; END LAYER 44
LIN {X -34.33, Y -49.21, Z 90.0, A 0, B 90, C 0} C_DIS
WAIT SEC 3
LIN {X -34.33, Y -49.21, Z 92.0, A 0, B 90, C 0} C_DIS
$OUT[1] = TRUE
WAIT SEC 0.8
LIN {X -34.33, Y -49.21, Z 92.0, A 0, B 90, C 0} C_DIS
LIN {X -34.33, Y -49.21, Z 92.0, A 0, B 90, C 0} C_DIS
LIN {X -31.75, Y -50.89, Z 92.0, A 0, B 90, C 0} C_DIS
LIN {X -31.1, Y -51.31, Z 92.0, A 0, B 90, C 0} C_DIS
LIN {X -28.42, Y -52.82, Z 92.0, A 0, B 90, C 0} C_DIS
LIN {X -27.75, Y -53.2, Z 92.0, A 0, B 90, C 0} C_DIS
LIN {X -24.98, Y -54.53, Z 92.0, A 0, B 90, C 0} C_DIS
LIN {X -24.29, Y -54.86, Z 92.0, A 0, B 90, C 0} C_DIS
LIN {X -21.43, Y -56.02, Z 92.0, A 0, B 90, C 0} C_DIS
LIN {X -20.72, Y -56.31, Z 92.0, A 0, B 90, C 0} C_DIS
LIN {X -17.8, Y -57.28, Z 92.0, A 0, B 90, C 0} C_DIS
LIN {X -17.07, Y -57.52, Z 92.0, A 0, B 90, C 0} C_DIS
LIN {X -14.1, Y -58.3, Z 92.0, A 0, B 90, C 0} C_DIS
LIN {X -13.35, Y -58.5, Z 92.0, A 0, B 90, C 0} C_DIS
LIN {X -10.33, Y -59.08, Z 92.0, A 0, B 90, C 0} C_DIS
LIN {X -9.58, Y -59.23, Z 92.0, A 0, B 90, C 0} C_DIS
LIN {X -6.52, Y -59.62, Z 92.0, A 0, B 90, C 0} C_DIS
LIN {X -5.76, Y -59.72, Z 92.0, A 0, B 90, C 0} C_DIS
LIN {X -2.69, Y -59.92, Z 92.0, A 0, B 90, C 0} C_DIS
LIN {X -1.92, Y -59.97, Z 92.0, A 0, B 90, C 0} C_DIS
LIN {X 1.15, Y -59.97, Z 92.0, A 0, B 90, C 0} C_DIS
LIN {X 1.92, Y -59.97, Z 92.0, A 0, B 90, C 0} C_DIS
LIN {X 4.99, Y -59.77, Z 92.0, A 0, B 90, C 0} C_DIS
LIN {X 5.76, Y -59.72, Z 92.0, A 0, B 90, C 0} C_DIS
LIN {X 8.81, Y -59.33, Z 92.0, A 0, B 90, C 0} C_DIS
LIN {X 9.58, Y -59.23, Z 92.0, A 0, B 90, C 0} C_DIS
LIN {X 12.6, Y -58.64, Z 92.0, A 0, B 90, C 0} C_DIS
LIN {X 13.35, Y -58.5, Z 92.0, A 0, B 90, C 0} C_DIS
LIN {X 16.33, Y -57.72, Z 92.0, A 0, B 90, C 0} C_DIS
LIN {X 17.07, Y -57.52, Z 92.0, A 0, B 90, C 0} C_DIS
LIN {X 19.99, Y -56.55, Z 92.0, A 0, B 90, C 0} C_DIS
LIN {X 20.72, Y -56.31, Z 92.0, A 0, B 90, C 0} C_DIS
LIN {X 23.57, Y -55.15, Z 92.0, A 0, B 90, C 0} C_DIS
LIN {X 24.29, Y -54.86, Z 92.0, A 0, B 90, C 0} C_DIS
LIN {X 27.06, Y -53.53, Z 92.0, A 0, B 90, C 0} C_DIS
LIN {X 27.75, Y -53.2, Z 92.0, A 0, B 90, C 0} C_DIS
LIN {X 30.43, Y -51.69, Z 92.0, A 0, B 90, C 0} C_DIS
LIN {X 31.1, Y -51.31, Z 92.0, A 0, B 90, C 0} C_DIS
LIN {X 33.68, Y -49.63, Z 92.0, A 0, B 90, C 0} C_DIS
LIN {X 34.33, Y -49.21, Z 92.0, A 0, B 90, C 0} C_DIS
LIN {X 36.79, Y -47.37, Z 92.0, A 0, B 90, C 0} C_DIS
LIN {X 37.41, Y -46.91, Z 92.0, A 0, B 90, C 0} C_DIS
LIN {X 39.75, Y -44.92, Z 92.0, A 0, B 90, C 0} C_DIS
LIN {X 40.34, Y -44.42, Z 92.0, A 0, B 90, C 0} C_DIS
LIN {X 42.55, Y -42.28, Z 92.0, A 0, B 90, C 0} C_DIS
LIN {X 43.1, Y -41.74, Z 92.0, A 0, B 90, C 0} C_DIS
LIN {X 45.17, Y -39.46, Z 92.0, A 0, B 90, C 0} C_DIS
LIN {X 45.69, Y -38.89, Z 92.0, A 0, B 90, C 0} C_DIS
LIN {X 47.61, Y -36.49, Z 92.0, A 0, B 90, C 0} C_DIS
LIN {X 48.08, Y -35.89, Z 92.0, A 0, B 90, C 0} C_DIS
LIN {X 49.85, Y -33.36, Z 92.0, A 0, B 90, C 0} C_DIS
LIN {X 50.29, Y -32.73, Z 92.0, A 0, B 90, C 0} C_DIS
LIN {X 51.88, Y -30.1, Z 92.0, A 0, B 90, C 0} C_DIS
LIN {X 52.28, Y -29.44, Z 92.0, A 0, B 90, C 0} C_DIS
LIN {X 53.7, Y -26.72, Z 92.0, A 0, B 90, C 0} C_DIS
LIN {X 54.06, Y -26.03, Z 92.0, A 0, B 90, C 0} C_DIS
LIN {X 55.3, Y -23.22, Z 92.0, A 0, B 90, C 0} C_DIS
LIN {X 55.62, Y -22.52, Z 92.0, A 0, B 90, C 0} C_DIS
LIN {X 56.68, Y -19.63, Z 92.0, A 0, B 90, C 0} C_DIS
LIN {X 56.94, Y -18.91, Z 92.0, A 0, B 90, C 0} C_DIS
LIN {X 57.82, Y -15.96, Z 92.0, A 0, B 90, C 0} C_DIS
LIN {X 58.04, Y -15.22, Z 92.0, A 0, B 90, C 0} C_DIS
LIN {X 58.72, Y -12.22, Z 92.0, A 0, B 90, C 0} C_DIS
LIN {X 58.89, Y -11.47, Z 92.0, A 0, B 90, C 0} C_DIS
LIN {X 59.38, Y -8.43, Z 92.0, A 0, B 90, C 0} C_DIS
LIN {X 59.51, Y -7.67, Z 92.0, A 0, B 90, C 0} C_DIS
LIN {X 59.8, Y -4.61, Z 92.0, A 0, B 90, C 0} C_DIS
LIN {X 59.88, Y -3.84, Z 92.0, A 0, B 90, C 0} C_DIS
LIN {X 59.98, Y -0.77, Z 92.0, A 0, B 90, C 0} C_DIS
LIN {X 60.0, Y -0.0, Z 92.0, A 0, B 90, C 0} C_DIS
LIN {X 59.9, Y 3.08, Z 92.0, A 0, B 90, C 0} C_DIS
LIN {X 59.88, Y 3.84, Z 92.0, A 0, B 90, C 0} C_DIS
LIN {X 59.58, Y 6.91, Z 92.0, A 0, B 90, C 0} C_DIS
LIN {X 59.51, Y 7.67, Z 92.0, A 0, B 90, C 0} C_DIS
LIN {X 59.02, Y 10.71, Z 92.0, A 0, B 90, C 0} C_DIS
LIN {X 58.89, Y 11.47, Z 92.0, A 0, B 90, C 0} C_DIS
LIN {X 58.21, Y 14.47, Z 92.0, A 0, B 90, C 0} C_DIS
LIN {X 58.04, Y 15.22, Z 92.0, A 0, B 90, C 0} C_DIS
LIN {X 57.16, Y 18.17, Z 92.0, A 0, B 90, C 0} C_DIS
LIN {X 56.94, Y 18.91, Z 92.0, A 0, B 90, C 0} C_DIS
LIN {X 55.88, Y 21.79, Z 92.0, A 0, B 90, C 0} C_DIS
LIN {X 55.62, Y 22.52, Z 92.0, A 0, B 90, C 0} C_DIS
LIN {X 54.37, Y 25.33, Z 92.0, A 0, B 90, C 0} C_DIS
LIN {X 54.06, Y 26.03, Z 92.0, A 0, B 90, C 0} C_DIS
LIN {X 52.63, Y 28.76, Z 92.0, A 0, B 90, C 0} C_DIS
LIN {X 52.28, Y 29.44, Z 92.0, A 0, B 90, C 0} C_DIS
LIN {X 50.68, Y 32.07, Z 92.0, A 0, B 90, C 0} C_DIS
LIN {X 50.29, Y 32.73, Z 92.0, A 0, B 90, C 0} C_DIS
LIN {X 48.52, Y 35.26, Z 92.0, A 0, B 90, C 0} C_DIS
LIN {X 48.08, Y 35.89, Z 92.0, A 0, B 90, C 0} C_DIS
LIN {X 46.17, Y 38.29, Z 92.0, A 0, B 90, C 0} C_DIS
LIN {X 45.69, Y 38.89, Z 92.0, A 0, B 90, C 0} C_DIS
LIN {X 43.62, Y 41.17, Z 92.0, A 0, B 90, C 0} C_DIS
LIN {X 43.1, Y 41.74, Z 92.0, A 0, B 90, C 0} C_DIS
LIN {X 40.89, Y 43.88, Z 92.0, A 0, B 90, C 0} C_DIS
LIN {X 40.34, Y 44.42, Z 92.0, A 0, B 90, C 0} C_DIS
LIN {X 38.0, Y 46.41, Z 92.0, A 0, B 90, C 0} C_DIS
LIN {X 37.41, Y 46.91, Z 92.0, A 0, B 90, C 0} C_DIS
LIN {X 34.94, Y 48.75, Z 92.0, A 0, B 90, C 0} C_DIS
LIN {X 34.33, Y 49.21, Z 92.0, A 0, B 90, C 0} C_DIS
LIN {X 31.75, Y 50.89, Z 92.0, A 0, B 90, C 0} C_DIS
LIN {X 31.1, Y 51.31, Z 92.0, A 0, B 90, C 0} C_DIS
LIN {X 28.42, Y 52.82, Z 92.0, A 0, B 90, C 0} C_DIS
LIN {X 27.75, Y 53.2, Z 92.0, A 0, B 90, C 0} C_DIS
LIN {X 24.98, Y 54.53, Z 92.0, A 0, B 90, C 0} C_DIS
LIN {X 24.29, Y 54.86, Z 92.0, A 0, B 90, C 0} C_DIS
LIN {X 21.43, Y 56.02, Z 92.0, A 0, B 90, C 0} C_DIS
LIN {X 20.72, Y 56.31, Z 92.0, A 0, B 90, C 0} C_DIS
LIN {X 17.8, Y 57.28, Z 92.0, A 0, B 90, C 0} C_DIS
LIN {X 17.07, Y 57.52, Z 92.0, A 0, B 90, C 0} C_DIS
LIN {X 14.1, Y 58.3, Z 92.0, A 0, B 90, C 0} C_DIS
LIN {X 13.35, Y 58.5, Z 92.0, A 0, B 90, C 0} C_DIS
LIN {X 10.33, Y 59.08, Z 92.0, A 0, B 90, C 0} C_DIS
LIN {X 9.58, Y 59.23, Z 92.0, A 0, B 90, C 0} C_DIS
LIN {X 6.52, Y 59.62, Z 92.0, A 0, B 90, C 0} C_DIS
LIN {X 5.76, Y 59.72, Z 92.0, A 0, B 90, C 0} C_DIS
LIN {X 2.69, Y 59.92, Z 92.0, A 0, B 90, C 0} C_DIS
LIN {X 1.92, Y 59.97, Z 92.0, A 0, B 90, C 0} C_DIS
LIN {X -1.15, Y 59.97, Z 92.0, A 0, B 90, C 0} C_DIS
LIN {X -1.92, Y 59.97, Z 92.0, A 0, B 90, C 0} C_DIS
LIN {X -4.99, Y 59.77, Z 92.0, A 0, B 90, C 0} C_DIS
LIN {X -5.76, Y 59.72, Z 92.0, A 0, B 90, C 0} C_DIS
LIN {X -8.81, Y 59.33, Z 92.0, A 0, B 90, C 0} C_DIS
LIN {X -9.58, Y 59.23, Z 92.0, A 0, B 90, C 0} C_DIS
LIN {X -12.6, Y 58.64, Z 92.0, A 0, B 90, C 0} C_DIS
LIN {X -13.35, Y 58.5, Z 92.0, A 0, B 90, C 0} C_DIS
LIN {X -16.33, Y 57.72, Z 92.0, A 0, B 90, C 0} C_DIS
LIN {X -17.07, Y 57.52, Z 92.0, A 0, B 90, C 0} C_DIS
LIN {X -19.99, Y 56.55, Z 92.0, A 0, B 90, C 0} C_DIS
LIN {X -20.72, Y 56.31, Z 92.0, A 0, B 90, C 0} C_DIS
LIN {X -23.57, Y 55.15, Z 92.0, A 0, B 90, C 0} C_DIS
LIN {X -24.29, Y 54.86, Z 92.0, A 0, B 90, C 0} C_DIS
LIN {X -27.06, Y 53.53, Z 92.0, A 0, B 90, C 0} C_DIS
LIN {X -27.75, Y 53.2, Z 92.0, A 0, B 90, C 0} C_DIS
LIN {X -30.43, Y 51.69, Z 92.0, A 0, B 90, C 0} C_DIS
LIN {X -31.1, Y 51.31, Z 92.0, A 0, B 90, C 0} C_DIS
LIN {X -33.68, Y 49.63, Z 92.0, A 0, B 90, C 0} C_DIS
LIN {X -34.33, Y 49.21, Z 92.0, A 0, B 90, C 0} C_DIS
LIN {X -36.79, Y 47.37, Z 92.0, A 0, B 90, C 0} C_DIS
LIN {X -37.41, Y 46.91, Z 92.0, A 0, B 90, C 0} C_DIS
LIN {X -39.75, Y 44.92, Z 92.0, A 0, B 90, C 0} C_DIS
LIN {X -40.34, Y 44.42, Z 92.0, A 0, B 90, C 0} C_DIS
LIN {X -42.55, Y 42.28, Z 92.0, A 0, B 90, C 0} C_DIS
LIN {X -43.1, Y 41.74, Z 92.0, A 0, B 90, C 0} C_DIS
LIN {X -45.17, Y 39.46, Z 92.0, A 0, B 90, C 0} C_DIS
LIN {X -45.69, Y 38.89, Z 92.0, A 0, B 90, C 0} C_DIS
LIN {X -47.61, Y 36.49, Z 92.0, A 0, B 90, C 0} C_DIS
LIN {X -48.08, Y 35.89, Z 92.0, A 0, B 90, C 0} C_DIS
LIN {X -49.85, Y 33.36, Z 92.0, A 0, B 90, C 0} C_DIS
LIN {X -50.29, Y 32.73, Z 92.0, A 0, B 90, C 0} C_DIS
LIN {X -51.88, Y 30.1, Z 92.0, A 0, B 90, C 0} C_DIS
LIN {X -52.28, Y 29.44, Z 92.0, A 0, B 90, C 0} C_DIS
LIN {X -53.7, Y 26.72, Z 92.0, A 0, B 90, C 0} C_DIS
LIN {X -54.06, Y 26.03, Z 92.0, A 0, B 90, C 0} C_DIS
LIN {X -55.3, Y 23.22, Z 92.0, A 0, B 90, C 0} C_DIS
LIN {X -55.62, Y 22.52, Z 92.0, A 0, B 90, C 0} C_DIS
LIN {X -56.68, Y 19.63, Z 92.0, A 0, B 90, C 0} C_DIS
LIN {X -56.94, Y 18.91, Z 92.0, A 0, B 90, C 0} C_DIS
LIN {X -57.82, Y 15.96, Z 92.0, A 0, B 90, C 0} C_DIS
LIN {X -58.04, Y 15.22, Z 92.0, A 0, B 90, C 0} C_DIS
LIN {X -58.72, Y 12.22, Z 92.0, A 0, B 90, C 0} C_DIS
LIN {X -58.89, Y 11.47, Z 92.0, A 0, B 90, C 0} C_DIS
LIN {X -59.38, Y 8.43, Z 92.0, A 0, B 90, C 0} C_DIS
LIN {X -59.51, Y 7.67, Z 92.0, A 0, B 90, C 0} C_DIS
LIN {X -59.8, Y 4.61, Z 92.0, A 0, B 90, C 0} C_DIS
LIN {X -59.88, Y 3.84, Z 92.0, A 0, B 90, C 0} C_DIS
LIN {X -59.98, Y 0.77, Z 92.0, A 0, B 90, C 0} C_DIS
LIN {X -60.0, Y -0.0, Z 92.0, A 0, B 90, C 0} C_DIS
LIN {X -59.9, Y -3.08, Z 92.0, A 0, B 90, C 0} C_DIS
LIN {X -59.88, Y -3.84, Z 92.0, A 0, B 90, C 0} C_DIS
LIN {X -59.58, Y -6.91, Z 92.0, A 0, B 90, C 0} C_DIS
LIN {X -59.51, Y -7.67, Z 92.0, A 0, B 90, C 0} C_DIS
LIN {X -59.02, Y -10.71, Z 92.0, A 0, B 90, C 0} C_DIS
LIN {X -58.89, Y -11.47, Z 92.0, A 0, B 90, C 0} C_DIS
LIN {X -58.21, Y -14.47, Z 92.0, A 0, B 90, C 0} C_DIS
LIN {X -58.04, Y -15.22, Z 92.0, A 0, B 90, C 0} C_DIS
LIN {X -57.16, Y -18.17, Z 92.0, A 0, B 90, C 0} C_DIS
LIN {X -56.94, Y -18.91, Z 92.0, A 0, B 90, C 0} C_DIS
LIN {X -55.88, Y -21.79, Z 92.0, A 0, B 90, C 0} C_DIS
LIN {X -55.62, Y -22.52, Z 92.0, A 0, B 90, C 0} C_DIS
LIN {X -54.37, Y -25.33, Z 92.0, A 0, B 90, C 0} C_DIS
LIN {X -54.06, Y -26.03, Z 92.0, A 0, B 90, C 0} C_DIS
LIN {X -52.63, Y -28.76, Z 92.0, A 0, B 90, C 0} C_DIS
LIN {X -52.28, Y -29.44, Z 92.0, A 0, B 90, C 0} C_DIS
LIN {X -50.68, Y -32.07, Z 92.0, A 0, B 90, C 0} C_DIS
LIN {X -50.29, Y -32.73, Z 92.0, A 0, B 90, C 0} C_DIS
LIN {X -48.52, Y -35.26, Z 92.0, A 0, B 90, C 0} C_DIS
LIN {X -48.08, Y -35.89, Z 92.0, A 0, B 90, C 0} C_DIS
LIN {X -46.17, Y -38.29, Z 92.0, A 0, B 90, C 0} C_DIS
LIN {X -45.69, Y -38.89, Z 92.0, A 0, B 90, C 0} C_DIS
LIN {X -43.62, Y -41.17, Z 92.0, A 0, B 90, C 0} C_DIS
LIN {X -43.1, Y -41.74, Z 92.0, A 0, B 90, C 0} C_DIS
LIN {X -40.89, Y -43.88, Z 92.0, A 0, B 90, C 0} C_DIS
LIN {X -40.34, Y -44.42, Z 92.0, A 0, B 90, C 0} C_DIS
LIN {X -38.0, Y -46.41, Z 92.0, A 0, B 90, C 0} C_DIS
LIN {X -37.41, Y -46.91, Z 92.0, A 0, B 90, C 0} C_DIS
LIN {X -34.94, Y -48.75, Z 92.0, A 0, B 90, C 0} C_DIS
$OUT[1] = FALSE

; END LAYER 45
LIN {X -34.33, Y -49.21, Z 92.0, A 0, B 90, C 0} C_DIS
WAIT SEC 3
LIN {X -34.33, Y -49.21, Z 94.0, A 0, B 90, C 0} C_DIS
$OUT[1] = TRUE
WAIT SEC 0.8
LIN {X -34.33, Y -49.21, Z 94.0, A 0, B 90, C 0} C_DIS
LIN {X -34.33, Y -49.21, Z 94.0, A 0, B 90, C 0} C_DIS
LIN {X -31.62, Y -50.97, Z 94.0, A 0, B 90, C 0} C_DIS
LIN {X -31.1, Y -51.31, Z 94.0, A 0, B 90, C 0} C_DIS
LIN {X -28.29, Y -52.89, Z 94.0, A 0, B 90, C 0} C_DIS
LIN {X -27.75, Y -53.2, Z 94.0, A 0, B 90, C 0} C_DIS
LIN {X -24.84, Y -54.6, Z 94.0, A 0, B 90, C 0} C_DIS
LIN {X -24.29, Y -54.86, Z 94.0, A 0, B 90, C 0} C_DIS
LIN {X -21.29, Y -56.08, Z 94.0, A 0, B 90, C 0} C_DIS
LIN {X -20.72, Y -56.31, Z 94.0, A 0, B 90, C 0} C_DIS
LIN {X -17.66, Y -57.33, Z 94.0, A 0, B 90, C 0} C_DIS
LIN {X -17.07, Y -57.52, Z 94.0, A 0, B 90, C 0} C_DIS
LIN {X -13.95, Y -58.34, Z 94.0, A 0, B 90, C 0} C_DIS
LIN {X -13.35, Y -58.5, Z 94.0, A 0, B 90, C 0} C_DIS
LIN {X -10.18, Y -59.11, Z 94.0, A 0, B 90, C 0} C_DIS
LIN {X -9.58, Y -59.23, Z 94.0, A 0, B 90, C 0} C_DIS
LIN {X -6.37, Y -59.64, Z 94.0, A 0, B 90, C 0} C_DIS
LIN {X -5.76, Y -59.72, Z 94.0, A 0, B 90, C 0} C_DIS
LIN {X -2.54, Y -59.93, Z 94.0, A 0, B 90, C 0} C_DIS
LIN {X -1.92, Y -59.97, Z 94.0, A 0, B 90, C 0} C_DIS
LIN {X 1.31, Y -59.97, Z 94.0, A 0, B 90, C 0} C_DIS
LIN {X 1.92, Y -59.97, Z 94.0, A 0, B 90, C 0} C_DIS
LIN {X 5.15, Y -59.76, Z 94.0, A 0, B 90, C 0} C_DIS
LIN {X 5.76, Y -59.72, Z 94.0, A 0, B 90, C 0} C_DIS
LIN {X 8.97, Y -59.31, Z 94.0, A 0, B 90, C 0} C_DIS
LIN {X 9.58, Y -59.23, Z 94.0, A 0, B 90, C 0} C_DIS
LIN {X 12.75, Y -58.61, Z 94.0, A 0, B 90, C 0} C_DIS
LIN {X 13.35, Y -58.5, Z 94.0, A 0, B 90, C 0} C_DIS
LIN {X 16.48, Y -57.68, Z 94.0, A 0, B 90, C 0} C_DIS
LIN {X 17.07, Y -57.52, Z 94.0, A 0, B 90, C 0} C_DIS
LIN {X 20.14, Y -56.5, Z 94.0, A 0, B 90, C 0} C_DIS
LIN {X 20.72, Y -56.31, Z 94.0, A 0, B 90, C 0} C_DIS
LIN {X 23.72, Y -55.1, Z 94.0, A 0, B 90, C 0} C_DIS
LIN {X 24.29, Y -54.86, Z 94.0, A 0, B 90, C 0} C_DIS
LIN {X 27.2, Y -53.46, Z 94.0, A 0, B 90, C 0} C_DIS
LIN {X 27.75, Y -53.2, Z 94.0, A 0, B 90, C 0} C_DIS
LIN {X 30.57, Y -51.61, Z 94.0, A 0, B 90, C 0} C_DIS
LIN {X 31.1, Y -51.31, Z 94.0, A 0, B 90, C 0} C_DIS
LIN {X 33.81, Y -49.55, Z 94.0, A 0, B 90, C 0} C_DIS
LIN {X 34.33, Y -49.21, Z 94.0, A 0, B 90, C 0} C_DIS
LIN {X 36.92, Y -47.28, Z 94.0, A 0, B 90, C 0} C_DIS
LIN {X 37.41, Y -46.91, Z 94.0, A 0, B 90, C 0} C_DIS
LIN {X 39.87, Y -44.82, Z 94.0, A 0, B 90, C 0} C_DIS
LIN {X 40.34, Y -44.42, Z 94.0, A 0, B 90, C 0} C_DIS
LIN {X 42.66, Y -42.17, Z 94.0, A 0, B 90, C 0} C_DIS
LIN {X 43.1, Y -41.74, Z 94.0, A 0, B 90, C 0} C_DIS
LIN {X 45.27, Y -39.35, Z 94.0, A 0, B 90, C 0} C_DIS
LIN {X 45.69, Y -38.89, Z 94.0, A 0, B 90, C 0} C_DIS
LIN {X 47.7, Y -36.37, Z 94.0, A 0, B 90, C 0} C_DIS
LIN {X 48.08, Y -35.89, Z 94.0, A 0, B 90, C 0} C_DIS
LIN {X 49.93, Y -33.24, Z 94.0, A 0, B 90, C 0} C_DIS
LIN {X 50.29, Y -32.73, Z 94.0, A 0, B 90, C 0} C_DIS
LIN {X 51.96, Y -29.97, Z 94.0, A 0, B 90, C 0} C_DIS
LIN {X 52.28, Y -29.44, Z 94.0, A 0, B 90, C 0} C_DIS
LIN {X 53.77, Y -26.58, Z 94.0, A 0, B 90, C 0} C_DIS
LIN {X 54.06, Y -26.03, Z 94.0, A 0, B 90, C 0} C_DIS
LIN {X 55.37, Y -23.08, Z 94.0, A 0, B 90, C 0} C_DIS
LIN {X 55.62, Y -22.52, Z 94.0, A 0, B 90, C 0} C_DIS
LIN {X 56.73, Y -19.48, Z 94.0, A 0, B 90, C 0} C_DIS
LIN {X 56.94, Y -18.91, Z 94.0, A 0, B 90, C 0} C_DIS
LIN {X 57.86, Y -15.81, Z 94.0, A 0, B 90, C 0} C_DIS
LIN {X 58.04, Y -15.22, Z 94.0, A 0, B 90, C 0} C_DIS
LIN {X 58.76, Y -12.07, Z 94.0, A 0, B 90, C 0} C_DIS
LIN {X 58.89, Y -11.47, Z 94.0, A 0, B 90, C 0} C_DIS
LIN {X 59.41, Y -8.28, Z 94.0, A 0, B 90, C 0} C_DIS
LIN {X 59.51, Y -7.67, Z 94.0, A 0, B 90, C 0} C_DIS
LIN {X 59.82, Y -4.46, Z 94.0, A 0, B 90, C 0} C_DIS
LIN {X 59.88, Y -3.84, Z 94.0, A 0, B 90, C 0} C_DIS
LIN {X 59.98, Y -0.62, Z 94.0, A 0, B 90, C 0} C_DIS
LIN {X 60.0, Y -0.0, Z 94.0, A 0, B 90, C 0} C_DIS
LIN {X 59.9, Y 3.23, Z 94.0, A 0, B 90, C 0} C_DIS
LIN {X 59.88, Y 3.84, Z 94.0, A 0, B 90, C 0} C_DIS
LIN {X 59.57, Y 7.06, Z 94.0, A 0, B 90, C 0} C_DIS
LIN {X 59.51, Y 7.67, Z 94.0, A 0, B 90, C 0} C_DIS
LIN {X 58.99, Y 10.86, Z 94.0, A 0, B 90, C 0} C_DIS
LIN {X 58.89, Y 11.47, Z 94.0, A 0, B 90, C 0} C_DIS
LIN {X 58.17, Y 14.62, Z 94.0, A 0, B 90, C 0} C_DIS
LIN {X 58.04, Y 15.22, Z 94.0, A 0, B 90, C 0} C_DIS
LIN {X 57.12, Y 18.32, Z 94.0, A 0, B 90, C 0} C_DIS
LIN {X 56.94, Y 18.91, Z 94.0, A 0, B 90, C 0} C_DIS
LIN {X 55.83, Y 21.94, Z 94.0, A 0, B 90, C 0} C_DIS
LIN {X 55.62, Y 22.52, Z 94.0, A 0, B 90, C 0} C_DIS
LIN {X 54.31, Y 25.47, Z 94.0, A 0, B 90, C 0} C_DIS
LIN {X 54.06, Y 26.03, Z 94.0, A 0, B 90, C 0} C_DIS
LIN {X 52.56, Y 28.9, Z 94.0, A 0, B 90, C 0} C_DIS
LIN {X 52.28, Y 29.44, Z 94.0, A 0, B 90, C 0} C_DIS
LIN {X 50.6, Y 32.21, Z 94.0, A 0, B 90, C 0} C_DIS
LIN {X 50.29, Y 32.73, Z 94.0, A 0, B 90, C 0} C_DIS
LIN {X 48.44, Y 35.38, Z 94.0, A 0, B 90, C 0} C_DIS
LIN {X 48.08, Y 35.89, Z 94.0, A 0, B 90, C 0} C_DIS
LIN {X 46.07, Y 38.41, Z 94.0, A 0, B 90, C 0} C_DIS
LIN {X 45.69, Y 38.89, Z 94.0, A 0, B 90, C 0} C_DIS
LIN {X 43.51, Y 41.29, Z 94.0, A 0, B 90, C 0} C_DIS
LIN {X 43.1, Y 41.74, Z 94.0, A 0, B 90, C 0} C_DIS
LIN {X 40.78, Y 43.99, Z 94.0, A 0, B 90, C 0} C_DIS
LIN {X 40.34, Y 44.42, Z 94.0, A 0, B 90, C 0} C_DIS
LIN {X 37.88, Y 46.51, Z 94.0, A 0, B 90, C 0} C_DIS
LIN {X 37.41, Y 46.91, Z 94.0, A 0, B 90, C 0} C_DIS
LIN {X 34.82, Y 48.84, Z 94.0, A 0, B 90, C 0} C_DIS
LIN {X 34.33, Y 49.21, Z 94.0, A 0, B 90, C 0} C_DIS
LIN {X 31.62, Y 50.97, Z 94.0, A 0, B 90, C 0} C_DIS
LIN {X 31.1, Y 51.31, Z 94.0, A 0, B 90, C 0} C_DIS
LIN {X 28.29, Y 52.89, Z 94.0, A 0, B 90, C 0} C_DIS
LIN {X 27.75, Y 53.2, Z 94.0, A 0, B 90, C 0} C_DIS
LIN {X 24.84, Y 54.6, Z 94.0, A 0, B 90, C 0} C_DIS
LIN {X 24.29, Y 54.86, Z 94.0, A 0, B 90, C 0} C_DIS
LIN {X 21.29, Y 56.08, Z 94.0, A 0, B 90, C 0} C_DIS
LIN {X 20.72, Y 56.31, Z 94.0, A 0, B 90, C 0} C_DIS
LIN {X 17.66, Y 57.33, Z 94.0, A 0, B 90, C 0} C_DIS
LIN {X 17.07, Y 57.52, Z 94.0, A 0, B 90, C 0} C_DIS
LIN {X 13.95, Y 58.34, Z 94.0, A 0, B 90, C 0} C_DIS
LIN {X 13.35, Y 58.5, Z 94.0, A 0, B 90, C 0} C_DIS
LIN {X 10.18, Y 59.11, Z 94.0, A 0, B 90, C 0} C_DIS
LIN {X 9.58, Y 59.23, Z 94.0, A 0, B 90, C 0} C_DIS
LIN {X 6.37, Y 59.64, Z 94.0, A 0, B 90, C 0} C_DIS
LIN {X 5.76, Y 59.72, Z 94.0, A 0, B 90, C 0} C_DIS
LIN {X 2.54, Y 59.93, Z 94.0, A 0, B 90, C 0} C_DIS
LIN {X 1.92, Y 59.97, Z 94.0, A 0, B 90, C 0} C_DIS
LIN {X -1.31, Y 59.97, Z 94.0, A 0, B 90, C 0} C_DIS
LIN {X -1.92, Y 59.97, Z 94.0, A 0, B 90, C 0} C_DIS
LIN {X -5.15, Y 59.76, Z 94.0, A 0, B 90, C 0} C_DIS
LIN {X -5.76, Y 59.72, Z 94.0, A 0, B 90, C 0} C_DIS
LIN {X -8.97, Y 59.31, Z 94.0, A 0, B 90, C 0} C_DIS
LIN {X -9.58, Y 59.23, Z 94.0, A 0, B 90, C 0} C_DIS
LIN {X -12.75, Y 58.61, Z 94.0, A 0, B 90, C 0} C_DIS
LIN {X -13.35, Y 58.5, Z 94.0, A 0, B 90, C 0} C_DIS
LIN {X -16.48, Y 57.68, Z 94.0, A 0, B 90, C 0} C_DIS
LIN {X -17.07, Y 57.52, Z 94.0, A 0, B 90, C 0} C_DIS
LIN {X -20.14, Y 56.5, Z 94.0, A 0, B 90, C 0} C_DIS
LIN {X -20.72, Y 56.31, Z 94.0, A 0, B 90, C 0} C_DIS
LIN {X -23.72, Y 55.1, Z 94.0, A 0, B 90, C 0} C_DIS
LIN {X -24.29, Y 54.86, Z 94.0, A 0, B 90, C 0} C_DIS
LIN {X -27.2, Y 53.46, Z 94.0, A 0, B 90, C 0} C_DIS
LIN {X -27.75, Y 53.2, Z 94.0, A 0, B 90, C 0} C_DIS
LIN {X -30.57, Y 51.61, Z 94.0, A 0, B 90, C 0} C_DIS
LIN {X -31.1, Y 51.31, Z 94.0, A 0, B 90, C 0} C_DIS
LIN {X -33.81, Y 49.55, Z 94.0, A 0, B 90, C 0} C_DIS
LIN {X -34.33, Y 49.21, Z 94.0, A 0, B 90, C 0} C_DIS
LIN {X -36.92, Y 47.28, Z 94.0, A 0, B 90, C 0} C_DIS
LIN {X -37.41, Y 46.91, Z 94.0, A 0, B 90, C 0} C_DIS
LIN {X -39.87, Y 44.82, Z 94.0, A 0, B 90, C 0} C_DIS
LIN {X -40.34, Y 44.42, Z 94.0, A 0, B 90, C 0} C_DIS
LIN {X -42.66, Y 42.17, Z 94.0, A 0, B 90, C 0} C_DIS
LIN {X -43.1, Y 41.74, Z 94.0, A 0, B 90, C 0} C_DIS
LIN {X -45.27, Y 39.35, Z 94.0, A 0, B 90, C 0} C_DIS
LIN {X -45.69, Y 38.89, Z 94.0, A 0, B 90, C 0} C_DIS
LIN {X -47.7, Y 36.37, Z 94.0, A 0, B 90, C 0} C_DIS
LIN {X -48.08, Y 35.89, Z 94.0, A 0, B 90, C 0} C_DIS
LIN {X -49.93, Y 33.24, Z 94.0, A 0, B 90, C 0} C_DIS
LIN {X -50.29, Y 32.73, Z 94.0, A 0, B 90, C 0} C_DIS
LIN {X -51.96, Y 29.97, Z 94.0, A 0, B 90, C 0} C_DIS
LIN {X -52.28, Y 29.44, Z 94.0, A 0, B 90, C 0} C_DIS
LIN {X -53.77, Y 26.58, Z 94.0, A 0, B 90, C 0} C_DIS
LIN {X -54.06, Y 26.03, Z 94.0, A 0, B 90, C 0} C_DIS
LIN {X -55.37, Y 23.08, Z 94.0, A 0, B 90, C 0} C_DIS
LIN {X -55.62, Y 22.52, Z 94.0, A 0, B 90, C 0} C_DIS
LIN {X -56.73, Y 19.48, Z 94.0, A 0, B 90, C 0} C_DIS
LIN {X -56.94, Y 18.91, Z 94.0, A 0, B 90, C 0} C_DIS
LIN {X -57.86, Y 15.81, Z 94.0, A 0, B 90, C 0} C_DIS
LIN {X -58.04, Y 15.22, Z 94.0, A 0, B 90, C 0} C_DIS
LIN {X -58.76, Y 12.07, Z 94.0, A 0, B 90, C 0} C_DIS
LIN {X -58.89, Y 11.47, Z 94.0, A 0, B 90, C 0} C_DIS
LIN {X -59.41, Y 8.28, Z 94.0, A 0, B 90, C 0} C_DIS
LIN {X -59.51, Y 7.67, Z 94.0, A 0, B 90, C 0} C_DIS
LIN {X -59.82, Y 4.46, Z 94.0, A 0, B 90, C 0} C_DIS
LIN {X -59.88, Y 3.84, Z 94.0, A 0, B 90, C 0} C_DIS
LIN {X -59.98, Y 0.62, Z 94.0, A 0, B 90, C 0} C_DIS
LIN {X -60.0, Y -0.0, Z 94.0, A 0, B 90, C 0} C_DIS
LIN {X -59.9, Y -3.23, Z 94.0, A 0, B 90, C 0} C_DIS
LIN {X -59.88, Y -3.84, Z 94.0, A 0, B 90, C 0} C_DIS
LIN {X -59.57, Y -7.06, Z 94.0, A 0, B 90, C 0} C_DIS
LIN {X -59.51, Y -7.67, Z 94.0, A 0, B 90, C 0} C_DIS
LIN {X -58.99, Y -10.86, Z 94.0, A 0, B 90, C 0} C_DIS
LIN {X -58.89, Y -11.47, Z 94.0, A 0, B 90, C 0} C_DIS
LIN {X -58.17, Y -14.62, Z 94.0, A 0, B 90, C 0} C_DIS
LIN {X -58.04, Y -15.22, Z 94.0, A 0, B 90, C 0} C_DIS
LIN {X -57.12, Y -18.32, Z 94.0, A 0, B 90, C 0} C_DIS
LIN {X -56.94, Y -18.91, Z 94.0, A 0, B 90, C 0} C_DIS
LIN {X -55.83, Y -21.94, Z 94.0, A 0, B 90, C 0} C_DIS
LIN {X -55.62, Y -22.52, Z 94.0, A 0, B 90, C 0} C_DIS
LIN {X -54.31, Y -25.47, Z 94.0, A 0, B 90, C 0} C_DIS
LIN {X -54.06, Y -26.03, Z 94.0, A 0, B 90, C 0} C_DIS
LIN {X -52.56, Y -28.9, Z 94.0, A 0, B 90, C 0} C_DIS
LIN {X -52.28, Y -29.44, Z 94.0, A 0, B 90, C 0} C_DIS
LIN {X -50.6, Y -32.21, Z 94.0, A 0, B 90, C 0} C_DIS
LIN {X -50.29, Y -32.73, Z 94.0, A 0, B 90, C 0} C_DIS
LIN {X -48.44, Y -35.38, Z 94.0, A 0, B 90, C 0} C_DIS
LIN {X -48.08, Y -35.89, Z 94.0, A 0, B 90, C 0} C_DIS
LIN {X -46.07, Y -38.41, Z 94.0, A 0, B 90, C 0} C_DIS
LIN {X -45.69, Y -38.89, Z 94.0, A 0, B 90, C 0} C_DIS
LIN {X -43.51, Y -41.29, Z 94.0, A 0, B 90, C 0} C_DIS
LIN {X -43.1, Y -41.74, Z 94.0, A 0, B 90, C 0} C_DIS
LIN {X -40.78, Y -43.99, Z 94.0, A 0, B 90, C 0} C_DIS
LIN {X -40.34, Y -44.42, Z 94.0, A 0, B 90, C 0} C_DIS
LIN {X -37.88, Y -46.51, Z 94.0, A 0, B 90, C 0} C_DIS
LIN {X -37.41, Y -46.91, Z 94.0, A 0, B 90, C 0} C_DIS
LIN {X -34.82, Y -48.84, Z 94.0, A 0, B 90, C 0} C_DIS
$OUT[1] = FALSE

; END LAYER 46
LIN {X -34.33, Y -49.21, Z 94.0, A 0, B 90, C 0} C_DIS
WAIT SEC 3
LIN {X -34.33, Y -49.21, Z 96.0, A 0, B 90, C 0} C_DIS
$OUT[1] = TRUE
WAIT SEC 0.8
LIN {X -34.33, Y -49.21, Z 96.0, A 0, B 90, C 0} C_DIS
LIN {X -34.33, Y -49.21, Z 96.0, A 0, B 90, C 0} C_DIS
LIN {X -31.49, Y -51.06, Z 96.0, A 0, B 90, C 0} C_DIS
LIN {X -31.1, Y -51.31, Z 96.0, A 0, B 90, C 0} C_DIS
LIN {X -28.15, Y -52.97, Z 96.0, A 0, B 90, C 0} C_DIS
LIN {X -27.75, Y -53.2, Z 96.0, A 0, B 90, C 0} C_DIS
LIN {X -24.7, Y -54.66, Z 96.0, A 0, B 90, C 0} C_DIS
LIN {X -24.29, Y -54.86, Z 96.0, A 0, B 90, C 0} C_DIS
LIN {X -21.15, Y -56.13, Z 96.0, A 0, B 90, C 0} C_DIS
LIN {X -20.72, Y -56.31, Z 96.0, A 0, B 90, C 0} C_DIS
LIN {X -17.51, Y -57.37, Z 96.0, A 0, B 90, C 0} C_DIS
LIN {X -17.07, Y -57.52, Z 96.0, A 0, B 90, C 0} C_DIS
LIN {X -13.8, Y -58.38, Z 96.0, A 0, B 90, C 0} C_DIS
LIN {X -13.35, Y -58.5, Z 96.0, A 0, B 90, C 0} C_DIS
LIN {X -10.03, Y -59.14, Z 96.0, A 0, B 90, C 0} C_DIS
LIN {X -9.58, Y -59.23, Z 96.0, A 0, B 90, C 0} C_DIS
LIN {X -6.22, Y -59.66, Z 96.0, A 0, B 90, C 0} C_DIS
LIN {X -5.76, Y -59.72, Z 96.0, A 0, B 90, C 0} C_DIS
LIN {X -2.38, Y -59.94, Z 96.0, A 0, B 90, C 0} C_DIS
LIN {X -1.92, Y -59.97, Z 96.0, A 0, B 90, C 0} C_DIS
LIN {X 1.46, Y -59.97, Z 96.0, A 0, B 90, C 0} C_DIS
LIN {X 1.92, Y -59.97, Z 96.0, A 0, B 90, C 0} C_DIS
LIN {X 5.3, Y -59.75, Z 96.0, A 0, B 90, C 0} C_DIS
LIN {X 5.76, Y -59.72, Z 96.0, A 0, B 90, C 0} C_DIS
LIN {X 9.12, Y -59.29, Z 96.0, A 0, B 90, C 0} C_DIS
LIN {X 9.58, Y -59.23, Z 96.0, A 0, B 90, C 0} C_DIS
LIN {X 12.9, Y -58.58, Z 96.0, A 0, B 90, C 0} C_DIS
LIN {X 13.35, Y -58.5, Z 96.0, A 0, B 90, C 0} C_DIS
LIN {X 16.63, Y -57.64, Z 96.0, A 0, B 90, C 0} C_DIS
LIN {X 17.07, Y -57.52, Z 96.0, A 0, B 90, C 0} C_DIS
LIN {X 20.28, Y -56.45, Z 96.0, A 0, B 90, C 0} C_DIS
LIN {X 20.72, Y -56.31, Z 96.0, A 0, B 90, C 0} C_DIS
LIN {X 23.86, Y -55.04, Z 96.0, A 0, B 90, C 0} C_DIS
LIN {X 24.29, Y -54.86, Z 96.0, A 0, B 90, C 0} C_DIS
LIN {X 27.34, Y -53.4, Z 96.0, A 0, B 90, C 0} C_DIS
LIN {X 27.75, Y -53.2, Z 96.0, A 0, B 90, C 0} C_DIS
LIN {X 30.7, Y -51.54, Z 96.0, A 0, B 90, C 0} C_DIS
LIN {X 31.1, Y -51.31, Z 96.0, A 0, B 90, C 0} C_DIS
LIN {X 33.94, Y -49.46, Z 96.0, A 0, B 90, C 0} C_DIS
LIN {X 34.33, Y -49.21, Z 96.0, A 0, B 90, C 0} C_DIS
LIN {X 37.04, Y -47.19, Z 96.0, A 0, B 90, C 0} C_DIS
LIN {X 37.41, Y -46.91, Z 96.0, A 0, B 90, C 0} C_DIS
LIN {X 39.99, Y -44.72, Z 96.0, A 0, B 90, C 0} C_DIS
LIN {X 40.34, Y -44.42, Z 96.0, A 0, B 90, C 0} C_DIS
LIN {X 42.77, Y -42.06, Z 96.0, A 0, B 90, C 0} C_DIS
LIN {X 43.1, Y -41.74, Z 96.0, A 0, B 90, C 0} C_DIS
LIN {X 45.38, Y -39.24, Z 96.0, A 0, B 90, C 0} C_DIS
LIN {X 45.69, Y -38.89, Z 96.0, A 0, B 90, C 0} C_DIS
LIN {X 47.8, Y -36.25, Z 96.0, A 0, B 90, C 0} C_DIS
LIN {X 48.08, Y -35.89, Z 96.0, A 0, B 90, C 0} C_DIS
LIN {X 50.02, Y -33.11, Z 96.0, A 0, B 90, C 0} C_DIS
LIN {X 50.29, Y -32.73, Z 96.0, A 0, B 90, C 0} C_DIS
LIN {X 52.04, Y -29.84, Z 96.0, A 0, B 90, C 0} C_DIS
LIN {X 52.28, Y -29.44, Z 96.0, A 0, B 90, C 0} C_DIS
LIN {X 53.84, Y -26.44, Z 96.0, A 0, B 90, C 0} C_DIS
LIN {X 54.06, Y -26.03, Z 96.0, A 0, B 90, C 0} C_DIS
LIN {X 55.43, Y -22.94, Z 96.0, A 0, B 90, C 0} C_DIS
LIN {X 55.62, Y -22.52, Z 96.0, A 0, B 90, C 0} C_DIS
LIN {X 56.78, Y -19.34, Z 96.0, A 0, B 90, C 0} C_DIS
LIN {X 56.94, Y -18.91, Z 96.0, A 0, B 90, C 0} C_DIS
LIN {X 57.91, Y -15.66, Z 96.0, A 0, B 90, C 0} C_DIS
LIN {X 58.04, Y -15.22, Z 96.0, A 0, B 90, C 0} C_DIS
LIN {X 58.79, Y -11.92, Z 96.0, A 0, B 90, C 0} C_DIS
LIN {X 58.89, Y -11.47, Z 96.0, A 0, B 90, C 0} C_DIS
LIN {X 59.43, Y -8.13, Z 96.0, A 0, B 90, C 0} C_DIS
LIN {X 59.51, Y -7.67, Z 96.0, A 0, B 90, C 0} C_DIS
LIN {X 59.83, Y -4.3, Z 96.0, A 0, B 90, C 0} C_DIS
LIN {X 59.88, Y -3.84, Z 96.0, A 0, B 90, C 0} C_DIS
LIN {X 59.99, Y -0.46, Z 96.0, A 0, B 90, C 0} C_DIS
LIN {X 60.0, Y 0.0, Z 96.0, A 0, B 90, C 0} C_DIS
LIN {X 59.89, Y 3.38, Z 96.0, A 0, B 90, C 0} C_DIS
LIN {X 59.88, Y 3.84, Z 96.0, A 0, B 90, C 0} C_DIS
LIN {X 59.55, Y 7.21, Z 96.0, A 0, B 90, C 0} C_DIS
LIN {X 59.51, Y 7.67, Z 96.0, A 0, B 90, C 0} C_DIS
LIN {X 58.97, Y 11.01, Z 96.0, A 0, B 90, C 0} C_DIS
LIN {X 58.89, Y 11.47, Z 96.0, A 0, B 90, C 0} C_DIS
LIN {X 58.14, Y 14.77, Z 96.0, A 0, B 90, C 0} C_DIS
LIN {X 58.04, Y 15.22, Z 96.0, A 0, B 90, C 0} C_DIS
LIN {X 57.07, Y 18.46, Z 96.0, A 0, B 90, C 0} C_DIS
LIN {X 56.94, Y 18.91, Z 96.0, A 0, B 90, C 0} C_DIS
LIN {X 55.77, Y 22.08, Z 96.0, A 0, B 90, C 0} C_DIS
LIN {X 55.62, Y 22.52, Z 96.0, A 0, B 90, C 0} C_DIS
LIN {X 54.24, Y 25.61, Z 96.0, A 0, B 90, C 0} C_DIS
LIN {X 54.06, Y 26.03, Z 96.0, A 0, B 90, C 0} C_DIS
LIN {X 52.49, Y 29.03, Z 96.0, A 0, B 90, C 0} C_DIS
LIN {X 52.28, Y 29.44, Z 96.0, A 0, B 90, C 0} C_DIS
LIN {X 50.52, Y 32.34, Z 96.0, A 0, B 90, C 0} C_DIS
LIN {X 50.29, Y 32.73, Z 96.0, A 0, B 90, C 0} C_DIS
LIN {X 48.35, Y 35.51, Z 96.0, A 0, B 90, C 0} C_DIS
LIN {X 48.08, Y 35.89, Z 96.0, A 0, B 90, C 0} C_DIS
LIN {X 45.97, Y 38.53, Z 96.0, A 0, B 90, C 0} C_DIS
LIN {X 45.69, Y 38.89, Z 96.0, A 0, B 90, C 0} C_DIS
LIN {X 43.41, Y 41.4, Z 96.0, A 0, B 90, C 0} C_DIS
LIN {X 43.1, Y 41.74, Z 96.0, A 0, B 90, C 0} C_DIS
LIN {X 40.67, Y 44.1, Z 96.0, A 0, B 90, C 0} C_DIS
LIN {X 40.34, Y 44.42, Z 96.0, A 0, B 90, C 0} C_DIS
LIN {X 37.76, Y 46.61, Z 96.0, A 0, B 90, C 0} C_DIS
LIN {X 37.41, Y 46.91, Z 96.0, A 0, B 90, C 0} C_DIS
LIN {X 34.7, Y 48.93, Z 96.0, A 0, B 90, C 0} C_DIS
LIN {X 34.33, Y 49.21, Z 96.0, A 0, B 90, C 0} C_DIS
LIN {X 31.49, Y 51.06, Z 96.0, A 0, B 90, C 0} C_DIS
LIN {X 31.1, Y 51.31, Z 96.0, A 0, B 90, C 0} C_DIS
LIN {X 28.15, Y 52.97, Z 96.0, A 0, B 90, C 0} C_DIS
LIN {X 27.75, Y 53.2, Z 96.0, A 0, B 90, C 0} C_DIS
LIN {X 24.7, Y 54.66, Z 96.0, A 0, B 90, C 0} C_DIS
LIN {X 24.29, Y 54.86, Z 96.0, A 0, B 90, C 0} C_DIS
LIN {X 21.15, Y 56.13, Z 96.0, A 0, B 90, C 0} C_DIS
LIN {X 20.72, Y 56.31, Z 96.0, A 0, B 90, C 0} C_DIS
LIN {X 17.51, Y 57.37, Z 96.0, A 0, B 90, C 0} C_DIS
LIN {X 17.07, Y 57.52, Z 96.0, A 0, B 90, C 0} C_DIS
LIN {X 13.8, Y 58.38, Z 96.0, A 0, B 90, C 0} C_DIS
LIN {X 13.35, Y 58.5, Z 96.0, A 0, B 90, C 0} C_DIS
LIN {X 10.03, Y 59.14, Z 96.0, A 0, B 90, C 0} C_DIS
LIN {X 9.58, Y 59.23, Z 96.0, A 0, B 90, C 0} C_DIS
LIN {X 6.22, Y 59.66, Z 96.0, A 0, B 90, C 0} C_DIS
LIN {X 5.76, Y 59.72, Z 96.0, A 0, B 90, C 0} C_DIS
LIN {X 2.38, Y 59.94, Z 96.0, A 0, B 90, C 0} C_DIS
LIN {X 1.92, Y 59.97, Z 96.0, A 0, B 90, C 0} C_DIS
LIN {X -1.46, Y 59.97, Z 96.0, A 0, B 90, C 0} C_DIS
LIN {X -1.92, Y 59.97, Z 96.0, A 0, B 90, C 0} C_DIS
LIN {X -5.3, Y 59.75, Z 96.0, A 0, B 90, C 0} C_DIS
LIN {X -5.76, Y 59.72, Z 96.0, A 0, B 90, C 0} C_DIS
LIN {X -9.12, Y 59.29, Z 96.0, A 0, B 90, C 0} C_DIS
LIN {X -9.58, Y 59.23, Z 96.0, A 0, B 90, C 0} C_DIS
LIN {X -12.9, Y 58.58, Z 96.0, A 0, B 90, C 0} C_DIS
LIN {X -13.35, Y 58.5, Z 96.0, A 0, B 90, C 0} C_DIS
LIN {X -16.63, Y 57.64, Z 96.0, A 0, B 90, C 0} C_DIS
LIN {X -17.07, Y 57.52, Z 96.0, A 0, B 90, C 0} C_DIS
LIN {X -20.28, Y 56.45, Z 96.0, A 0, B 90, C 0} C_DIS
LIN {X -20.72, Y 56.31, Z 96.0, A 0, B 90, C 0} C_DIS
LIN {X -23.86, Y 55.04, Z 96.0, A 0, B 90, C 0} C_DIS
LIN {X -24.29, Y 54.86, Z 96.0, A 0, B 90, C 0} C_DIS
LIN {X -27.34, Y 53.4, Z 96.0, A 0, B 90, C 0} C_DIS
LIN {X -27.75, Y 53.2, Z 96.0, A 0, B 90, C 0} C_DIS
LIN {X -30.7, Y 51.54, Z 96.0, A 0, B 90, C 0} C_DIS
LIN {X -31.1, Y 51.31, Z 96.0, A 0, B 90, C 0} C_DIS
LIN {X -33.94, Y 49.46, Z 96.0, A 0, B 90, C 0} C_DIS
LIN {X -34.33, Y 49.21, Z 96.0, A 0, B 90, C 0} C_DIS
LIN {X -37.04, Y 47.19, Z 96.0, A 0, B 90, C 0} C_DIS
LIN {X -37.41, Y 46.91, Z 96.0, A 0, B 90, C 0} C_DIS
LIN {X -39.99, Y 44.72, Z 96.0, A 0, B 90, C 0} C_DIS
LIN {X -40.34, Y 44.42, Z 96.0, A 0, B 90, C 0} C_DIS
LIN {X -42.77, Y 42.06, Z 96.0, A 0, B 90, C 0} C_DIS
LIN {X -43.1, Y 41.74, Z 96.0, A 0, B 90, C 0} C_DIS
LIN {X -45.38, Y 39.24, Z 96.0, A 0, B 90, C 0} C_DIS
LIN {X -45.69, Y 38.89, Z 96.0, A 0, B 90, C 0} C_DIS
LIN {X -47.8, Y 36.25, Z 96.0, A 0, B 90, C 0} C_DIS
LIN {X -48.08, Y 35.89, Z 96.0, A 0, B 90, C 0} C_DIS
LIN {X -50.02, Y 33.11, Z 96.0, A 0, B 90, C 0} C_DIS
LIN {X -50.29, Y 32.73, Z 96.0, A 0, B 90, C 0} C_DIS
LIN {X -52.04, Y 29.84, Z 96.0, A 0, B 90, C 0} C_DIS
LIN {X -52.28, Y 29.44, Z 96.0, A 0, B 90, C 0} C_DIS
LIN {X -53.84, Y 26.44, Z 96.0, A 0, B 90, C 0} C_DIS
LIN {X -54.06, Y 26.03, Z 96.0, A 0, B 90, C 0} C_DIS
LIN {X -55.43, Y 22.94, Z 96.0, A 0, B 90, C 0} C_DIS
LIN {X -55.62, Y 22.52, Z 96.0, A 0, B 90, C 0} C_DIS
LIN {X -56.78, Y 19.34, Z 96.0, A 0, B 90, C 0} C_DIS
LIN {X -56.94, Y 18.91, Z 96.0, A 0, B 90, C 0} C_DIS
LIN {X -57.91, Y 15.66, Z 96.0, A 0, B 90, C 0} C_DIS
LIN {X -58.04, Y 15.22, Z 96.0, A 0, B 90, C 0} C_DIS
LIN {X -58.79, Y 11.92, Z 96.0, A 0, B 90, C 0} C_DIS
LIN {X -58.89, Y 11.47, Z 96.0, A 0, B 90, C 0} C_DIS
LIN {X -59.43, Y 8.13, Z 96.0, A 0, B 90, C 0} C_DIS
LIN {X -59.51, Y 7.67, Z 96.0, A 0, B 90, C 0} C_DIS
LIN {X -59.83, Y 4.3, Z 96.0, A 0, B 90, C 0} C_DIS
LIN {X -59.88, Y 3.84, Z 96.0, A 0, B 90, C 0} C_DIS
LIN {X -59.99, Y 0.46, Z 96.0, A 0, B 90, C 0} C_DIS
LIN {X -60.0, Y -0.0, Z 96.0, A 0, B 90, C 0} C_DIS
LIN {X -59.89, Y -3.38, Z 96.0, A 0, B 90, C 0} C_DIS
LIN {X -59.88, Y -3.84, Z 96.0, A 0, B 90, C 0} C_DIS
LIN {X -59.55, Y -7.21, Z 96.0, A 0, B 90, C 0} C_DIS
LIN {X -59.51, Y -7.67, Z 96.0, A 0, B 90, C 0} C_DIS
LIN {X -58.97, Y -11.01, Z 96.0, A 0, B 90, C 0} C_DIS
LIN {X -58.89, Y -11.47, Z 96.0, A 0, B 90, C 0} C_DIS
LIN {X -58.14, Y -14.77, Z 96.0, A 0, B 90, C 0} C_DIS
LIN {X -58.04, Y -15.22, Z 96.0, A 0, B 90, C 0} C_DIS
LIN {X -57.07, Y -18.46, Z 96.0, A 0, B 90, C 0} C_DIS
LIN {X -56.94, Y -18.91, Z 96.0, A 0, B 90, C 0} C_DIS
LIN {X -55.77, Y -22.08, Z 96.0, A 0, B 90, C 0} C_DIS
LIN {X -55.62, Y -22.52, Z 96.0, A 0, B 90, C 0} C_DIS
LIN {X -54.24, Y -25.61, Z 96.0, A 0, B 90, C 0} C_DIS
LIN {X -54.06, Y -26.03, Z 96.0, A 0, B 90, C 0} C_DIS
LIN {X -52.49, Y -29.03, Z 96.0, A 0, B 90, C 0} C_DIS
LIN {X -52.28, Y -29.44, Z 96.0, A 0, B 90, C 0} C_DIS
LIN {X -50.52, Y -32.34, Z 96.0, A 0, B 90, C 0} C_DIS
LIN {X -50.29, Y -32.73, Z 96.0, A 0, B 90, C 0} C_DIS
LIN {X -48.35, Y -35.51, Z 96.0, A 0, B 90, C 0} C_DIS
LIN {X -48.08, Y -35.89, Z 96.0, A 0, B 90, C 0} C_DIS
LIN {X -45.97, Y -38.53, Z 96.0, A 0, B 90, C 0} C_DIS
LIN {X -45.69, Y -38.89, Z 96.0, A 0, B 90, C 0} C_DIS
LIN {X -43.41, Y -41.4, Z 96.0, A 0, B 90, C 0} C_DIS
LIN {X -43.1, Y -41.74, Z 96.0, A 0, B 90, C 0} C_DIS
LIN {X -40.67, Y -44.1, Z 96.0, A 0, B 90, C 0} C_DIS
LIN {X -40.34, Y -44.42, Z 96.0, A 0, B 90, C 0} C_DIS
LIN {X -37.76, Y -46.61, Z 96.0, A 0, B 90, C 0} C_DIS
LIN {X -37.41, Y -46.91, Z 96.0, A 0, B 90, C 0} C_DIS
LIN {X -34.7, Y -48.93, Z 96.0, A 0, B 90, C 0} C_DIS
$OUT[1] = FALSE

; END LAYER 47
LIN {X -34.33, Y -49.21, Z 96.0, A 0, B 90, C 0} C_DIS
WAIT SEC 3
LIN {X -34.33, Y -49.21, Z 98.0, A 0, B 90, C 0} C_DIS
$OUT[1] = TRUE
WAIT SEC 0.8
LIN {X -34.33, Y -49.21, Z 98.0, A 0, B 90, C 0} C_DIS
LIN {X -34.33, Y -49.21, Z 98.0, A 0, B 90, C 0} C_DIS
LIN {X -31.36, Y -51.14, Z 98.0, A 0, B 90, C 0} C_DIS
LIN {X -31.1, Y -51.31, Z 98.0, A 0, B 90, C 0} C_DIS
LIN {X -28.02, Y -53.04, Z 98.0, A 0, B 90, C 0} C_DIS
LIN {X -27.75, Y -53.2, Z 98.0, A 0, B 90, C 0} C_DIS
LIN {X -24.56, Y -54.73, Z 98.0, A 0, B 90, C 0} C_DIS
LIN {X -24.29, Y -54.86, Z 98.0, A 0, B 90, C 0} C_DIS
LIN {X -21.01, Y -56.19, Z 98.0, A 0, B 90, C 0} C_DIS
LIN {X -20.72, Y -56.31, Z 98.0, A 0, B 90, C 0} C_DIS
LIN {X -17.36, Y -57.42, Z 98.0, A 0, B 90, C 0} C_DIS
LIN {X -17.07, Y -57.52, Z 98.0, A 0, B 90, C 0} C_DIS
LIN {X -13.65, Y -58.42, Z 98.0, A 0, B 90, C 0} C_DIS
LIN {X -13.35, Y -58.5, Z 98.0, A 0, B 90, C 0} C_DIS
LIN {X -9.88, Y -59.17, Z 98.0, A 0, B 90, C 0} C_DIS
LIN {X -9.58, Y -59.23, Z 98.0, A 0, B 90, C 0} C_DIS
LIN {X -6.07, Y -59.68, Z 98.0, A 0, B 90, C 0} C_DIS
LIN {X -5.76, Y -59.72, Z 98.0, A 0, B 90, C 0} C_DIS
LIN {X -2.23, Y -59.95, Z 98.0, A 0, B 90, C 0} C_DIS
LIN {X -1.92, Y -59.97, Z 98.0, A 0, B 90, C 0} C_DIS
LIN {X 1.62, Y -59.97, Z 98.0, A 0, B 90, C 0} C_DIS
LIN {X 1.92, Y -59.97, Z 98.0, A 0, B 90, C 0} C_DIS
LIN {X 5.45, Y -59.74, Z 98.0, A 0, B 90, C 0} C_DIS
LIN {X 5.76, Y -59.72, Z 98.0, A 0, B 90, C 0} C_DIS
LIN {X 9.27, Y -59.27, Z 98.0, A 0, B 90, C 0} C_DIS
LIN {X 9.58, Y -59.23, Z 98.0, A 0, B 90, C 0} C_DIS
LIN {X 13.05, Y -58.55, Z 98.0, A 0, B 90, C 0} C_DIS
LIN {X 13.35, Y -58.5, Z 98.0, A 0, B 90, C 0} C_DIS
LIN {X 16.77, Y -57.6, Z 98.0, A 0, B 90, C 0} C_DIS
LIN {X 17.07, Y -57.52, Z 98.0, A 0, B 90, C 0} C_DIS
LIN {X 20.43, Y -56.41, Z 98.0, A 0, B 90, C 0} C_DIS
LIN {X 20.72, Y -56.31, Z 98.0, A 0, B 90, C 0} C_DIS
LIN {X 24.0, Y -54.98, Z 98.0, A 0, B 90, C 0} C_DIS
LIN {X 24.29, Y -54.86, Z 98.0, A 0, B 90, C 0} C_DIS
LIN {X 27.48, Y -53.33, Z 98.0, A 0, B 90, C 0} C_DIS
LIN {X 27.75, Y -53.2, Z 98.0, A 0, B 90, C 0} C_DIS
LIN {X 30.84, Y -51.46, Z 98.0, A 0, B 90, C 0} C_DIS
LIN {X 31.1, Y -51.31, Z 98.0, A 0, B 90, C 0} C_DIS
LIN {X 34.07, Y -49.38, Z 98.0, A 0, B 90, C 0} C_DIS
LIN {X 34.33, Y -49.21, Z 98.0, A 0, B 90, C 0} C_DIS
LIN {X 37.16, Y -47.09, Z 98.0, A 0, B 90, C 0} C_DIS
LIN {X 37.41, Y -46.91, Z 98.0, A 0, B 90, C 0} C_DIS
LIN {X 40.1, Y -44.62, Z 98.0, A 0, B 90, C 0} C_DIS
LIN {X 40.34, Y -44.42, Z 98.0, A 0, B 90, C 0} C_DIS
LIN {X 42.88, Y -41.96, Z 98.0, A 0, B 90, C 0} C_DIS
LIN {X 43.1, Y -41.74, Z 98.0, A 0, B 90, C 0} C_DIS
LIN {X 45.48, Y -39.12, Z 98.0, A 0, B 90, C 0} C_DIS
LIN {X 45.69, Y -38.89, Z 98.0, A 0, B 90, C 0} C_DIS
LIN {X 47.89, Y -36.13, Z 98.0, A 0, B 90, C 0} C_DIS
LIN {X 48.08, Y -35.89, Z 98.0, A 0, B 90, C 0} C_DIS
LIN {X 50.11, Y -32.98, Z 98.0, A 0, B 90, C 0} C_DIS
LIN {X 50.29, Y -32.73, Z 98.0, A 0, B 90, C 0} C_DIS
LIN {X 52.12, Y -29.71, Z 98.0, A 0, B 90, C 0} C_DIS
LIN {X 52.28, Y -29.44, Z 98.0, A 0, B 90, C 0} C_DIS
LIN {X 53.92, Y -26.31, Z 98.0, A 0, B 90, C 0} C_DIS
LIN {X 54.06, Y -26.03, Z 98.0, A 0, B 90, C 0} C_DIS
LIN {X 55.49, Y -22.8, Z 98.0, A 0, B 90, C 0} C_DIS
LIN {X 55.62, Y -22.52, Z 98.0, A 0, B 90, C 0} C_DIS
LIN {X 56.84, Y -19.2, Z 98.0, A 0, B 90, C 0} C_DIS
LIN {X 56.94, Y -18.91, Z 98.0, A 0, B 90, C 0} C_DIS
LIN {X 57.95, Y -15.51, Z 98.0, A 0, B 90, C 0} C_DIS
LIN {X 58.04, Y -15.22, Z 98.0, A 0, B 90, C 0} C_DIS
LIN {X 58.83, Y -11.77, Z 98.0, A 0, B 90, C 0} C_DIS
LIN {X 58.89, Y -11.47, Z 98.0, A 0, B 90, C 0} C_DIS
LIN {X 59.46, Y -7.98, Z 98.0, A 0, B 90, C 0} C_DIS
LIN {X 59.51, Y -7.67, Z 98.0, A 0, B 90, C 0} C_DIS
LIN {X 59.85, Y -4.15, Z 98.0, A 0, B 90, C 0} C_DIS
LIN {X 59.88, Y -3.84, Z 98.0, A 0, B 90, C 0} C_DIS
LIN {X 59.99, Y -0.31, Z 98.0, A 0, B 90, C 0} C_DIS
LIN {X 60.0, Y -0.0, Z 98.0, A 0, B 90, C 0} C_DIS
LIN {X 59.89, Y 3.54, Z 98.0, A 0, B 90, C 0} C_DIS
LIN {X 59.88, Y 3.84, Z 98.0, A 0, B 90, C 0} C_DIS
LIN {X 59.54, Y 7.37, Z 98.0, A 0, B 90, C 0} C_DIS
LIN {X 59.51, Y 7.67, Z 98.0, A 0, B 90, C 0} C_DIS
LIN {X 58.94, Y 11.17, Z 98.0, A 0, B 90, C 0} C_DIS
LIN {X 58.89, Y 11.47, Z 98.0, A 0, B 90, C 0} C_DIS
LIN {X 58.11, Y 14.92, Z 98.0, A 0, B 90, C 0} C_DIS
LIN {X 58.04, Y 15.22, Z 98.0, A 0, B 90, C 0} C_DIS
LIN {X 57.03, Y 18.61, Z 98.0, A 0, B 90, C 0} C_DIS
LIN {X 56.94, Y 18.91, Z 98.0, A 0, B 90, C 0} C_DIS
LIN {X 55.72, Y 22.23, Z 98.0, A 0, B 90, C 0} C_DIS
LIN {X 55.62, Y 22.52, Z 98.0, A 0, B 90, C 0} C_DIS
LIN {X 54.18, Y 25.75, Z 98.0, A 0, B 90, C 0} C_DIS
LIN {X 54.06, Y 26.03, Z 98.0, A 0, B 90, C 0} C_DIS
LIN {X 52.42, Y 29.17, Z 98.0, A 0, B 90, C 0} C_DIS
LIN {X 52.28, Y 29.44, Z 98.0, A 0, B 90, C 0} C_DIS
LIN {X 50.44, Y 32.47, Z 98.0, A 0, B 90, C 0} C_DIS
LIN {X 50.29, Y 32.73, Z 98.0, A 0, B 90, C 0} C_DIS
LIN {X 48.26, Y 35.63, Z 98.0, A 0, B 90, C 0} C_DIS
LIN {X 48.08, Y 35.89, Z 98.0, A 0, B 90, C 0} C_DIS
LIN {X 45.88, Y 38.65, Z 98.0, A 0, B 90, C 0} C_DIS
LIN {X 45.69, Y 38.89, Z 98.0, A 0, B 90, C 0} C_DIS
LIN {X 43.31, Y 41.51, Z 98.0, A 0, B 90, C 0} C_DIS
LIN {X 43.1, Y 41.74, Z 98.0, A 0, B 90, C 0} C_DIS
LIN {X 40.56, Y 44.2, Z 98.0, A 0, B 90, C 0} C_DIS
LIN {X 40.34, Y 44.42, Z 98.0, A 0, B 90, C 0} C_DIS
LIN {X 37.64, Y 46.71, Z 98.0, A 0, B 90, C 0} C_DIS
LIN {X 37.41, Y 46.91, Z 98.0, A 0, B 90, C 0} C_DIS
LIN {X 34.57, Y 49.03, Z 98.0, A 0, B 90, C 0} C_DIS
LIN {X 34.33, Y 49.21, Z 98.0, A 0, B 90, C 0} C_DIS
LIN {X 31.36, Y 51.14, Z 98.0, A 0, B 90, C 0} C_DIS
LIN {X 31.1, Y 51.31, Z 98.0, A 0, B 90, C 0} C_DIS
LIN {X 28.02, Y 53.04, Z 98.0, A 0, B 90, C 0} C_DIS
LIN {X 27.75, Y 53.2, Z 98.0, A 0, B 90, C 0} C_DIS
LIN {X 24.56, Y 54.73, Z 98.0, A 0, B 90, C 0} C_DIS
LIN {X 24.29, Y 54.86, Z 98.0, A 0, B 90, C 0} C_DIS
LIN {X 21.01, Y 56.19, Z 98.0, A 0, B 90, C 0} C_DIS
LIN {X 20.72, Y 56.31, Z 98.0, A 0, B 90, C 0} C_DIS
LIN {X 17.36, Y 57.42, Z 98.0, A 0, B 90, C 0} C_DIS
LIN {X 17.07, Y 57.52, Z 98.0, A 0, B 90, C 0} C_DIS
LIN {X 13.65, Y 58.42, Z 98.0, A 0, B 90, C 0} C_DIS
LIN {X 13.35, Y 58.5, Z 98.0, A 0, B 90, C 0} C_DIS
LIN {X 9.88, Y 59.17, Z 98.0, A 0, B 90, C 0} C_DIS
LIN {X 9.58, Y 59.23, Z 98.0, A 0, B 90, C 0} C_DIS
LIN {X 6.07, Y 59.68, Z 98.0, A 0, B 90, C 0} C_DIS
LIN {X 5.76, Y 59.72, Z 98.0, A 0, B 90, C 0} C_DIS
LIN {X 2.23, Y 59.95, Z 98.0, A 0, B 90, C 0} C_DIS
LIN {X 1.92, Y 59.97, Z 98.0, A 0, B 90, C 0} C_DIS
LIN {X -1.62, Y 59.97, Z 98.0, A 0, B 90, C 0} C_DIS
LIN {X -1.92, Y 59.97, Z 98.0, A 0, B 90, C 0} C_DIS
LIN {X -5.45, Y 59.74, Z 98.0, A 0, B 90, C 0} C_DIS
LIN {X -5.76, Y 59.72, Z 98.0, A 0, B 90, C 0} C_DIS
LIN {X -9.27, Y 59.27, Z 98.0, A 0, B 90, C 0} C_DIS
LIN {X -9.58, Y 59.23, Z 98.0, A 0, B 90, C 0} C_DIS
LIN {X -13.05, Y 58.55, Z 98.0, A 0, B 90, C 0} C_DIS
LIN {X -13.35, Y 58.5, Z 98.0, A 0, B 90, C 0} C_DIS
LIN {X -16.77, Y 57.6, Z 98.0, A 0, B 90, C 0} C_DIS
LIN {X -17.07, Y 57.52, Z 98.0, A 0, B 90, C 0} C_DIS
LIN {X -20.43, Y 56.41, Z 98.0, A 0, B 90, C 0} C_DIS
LIN {X -20.72, Y 56.31, Z 98.0, A 0, B 90, C 0} C_DIS
LIN {X -24.0, Y 54.98, Z 98.0, A 0, B 90, C 0} C_DIS
LIN {X -24.29, Y 54.86, Z 98.0, A 0, B 90, C 0} C_DIS
LIN {X -27.48, Y 53.33, Z 98.0, A 0, B 90, C 0} C_DIS
LIN {X -27.75, Y 53.2, Z 98.0, A 0, B 90, C 0} C_DIS
LIN {X -30.84, Y 51.46, Z 98.0, A 0, B 90, C 0} C_DIS
LIN {X -31.1, Y 51.31, Z 98.0, A 0, B 90, C 0} C_DIS
LIN {X -34.07, Y 49.38, Z 98.0, A 0, B 90, C 0} C_DIS
LIN {X -34.33, Y 49.21, Z 98.0, A 0, B 90, C 0} C_DIS
LIN {X -37.16, Y 47.09, Z 98.0, A 0, B 90, C 0} C_DIS
LIN {X -37.41, Y 46.91, Z 98.0, A 0, B 90, C 0} C_DIS
LIN {X -40.1, Y 44.62, Z 98.0, A 0, B 90, C 0} C_DIS
LIN {X -40.34, Y 44.42, Z 98.0, A 0, B 90, C 0} C_DIS
LIN {X -42.88, Y 41.96, Z 98.0, A 0, B 90, C 0} C_DIS
LIN {X -43.1, Y 41.74, Z 98.0, A 0, B 90, C 0} C_DIS
LIN {X -45.48, Y 39.12, Z 98.0, A 0, B 90, C 0} C_DIS
LIN {X -45.69, Y 38.89, Z 98.0, A 0, B 90, C 0} C_DIS
LIN {X -47.89, Y 36.13, Z 98.0, A 0, B 90, C 0} C_DIS
LIN {X -48.08, Y 35.89, Z 98.0, A 0, B 90, C 0} C_DIS
LIN {X -50.11, Y 32.98, Z 98.0, A 0, B 90, C 0} C_DIS
LIN {X -50.29, Y 32.73, Z 98.0, A 0, B 90, C 0} C_DIS
LIN {X -52.12, Y 29.71, Z 98.0, A 0, B 90, C 0} C_DIS
LIN {X -52.28, Y 29.44, Z 98.0, A 0, B 90, C 0} C_DIS
LIN {X -53.92, Y 26.31, Z 98.0, A 0, B 90, C 0} C_DIS
LIN {X -54.06, Y 26.03, Z 98.0, A 0, B 90, C 0} C_DIS
LIN {X -55.49, Y 22.8, Z 98.0, A 0, B 90, C 0} C_DIS
LIN {X -55.62, Y 22.52, Z 98.0, A 0, B 90, C 0} C_DIS
LIN {X -56.84, Y 19.2, Z 98.0, A 0, B 90, C 0} C_DIS
LIN {X -56.94, Y 18.91, Z 98.0, A 0, B 90, C 0} C_DIS
LIN {X -57.95, Y 15.51, Z 98.0, A 0, B 90, C 0} C_DIS
LIN {X -58.04, Y 15.22, Z 98.0, A 0, B 90, C 0} C_DIS
LIN {X -58.83, Y 11.77, Z 98.0, A 0, B 90, C 0} C_DIS
LIN {X -58.89, Y 11.47, Z 98.0, A 0, B 90, C 0} C_DIS
LIN {X -59.46, Y 7.98, Z 98.0, A 0, B 90, C 0} C_DIS
LIN {X -59.51, Y 7.67, Z 98.0, A 0, B 90, C 0} C_DIS
LIN {X -59.85, Y 4.15, Z 98.0, A 0, B 90, C 0} C_DIS
LIN {X -59.88, Y 3.84, Z 98.0, A 0, B 90, C 0} C_DIS
LIN {X -59.99, Y 0.31, Z 98.0, A 0, B 90, C 0} C_DIS
LIN {X -60.0, Y -0.0, Z 98.0, A 0, B 90, C 0} C_DIS
LIN {X -59.89, Y -3.54, Z 98.0, A 0, B 90, C 0} C_DIS
LIN {X -59.88, Y -3.84, Z 98.0, A 0, B 90, C 0} C_DIS
LIN {X -59.54, Y -7.37, Z 98.0, A 0, B 90, C 0} C_DIS
LIN {X -59.51, Y -7.67, Z 98.0, A 0, B 90, C 0} C_DIS
LIN {X -58.94, Y -11.17, Z 98.0, A 0, B 90, C 0} C_DIS
LIN {X -58.89, Y -11.47, Z 98.0, A 0, B 90, C 0} C_DIS
LIN {X -58.11, Y -14.92, Z 98.0, A 0, B 90, C 0} C_DIS
LIN {X -58.04, Y -15.22, Z 98.0, A 0, B 90, C 0} C_DIS
LIN {X -57.03, Y -18.61, Z 98.0, A 0, B 90, C 0} C_DIS
LIN {X -56.94, Y -18.91, Z 98.0, A 0, B 90, C 0} C_DIS
LIN {X -55.72, Y -22.23, Z 98.0, A 0, B 90, C 0} C_DIS
LIN {X -55.62, Y -22.52, Z 98.0, A 0, B 90, C 0} C_DIS
LIN {X -54.18, Y -25.75, Z 98.0, A 0, B 90, C 0} C_DIS
LIN {X -54.06, Y -26.03, Z 98.0, A 0, B 90, C 0} C_DIS
LIN {X -52.42, Y -29.17, Z 98.0, A 0, B 90, C 0} C_DIS
LIN {X -52.28, Y -29.44, Z 98.0, A 0, B 90, C 0} C_DIS
LIN {X -50.44, Y -32.47, Z 98.0, A 0, B 90, C 0} C_DIS
LIN {X -50.29, Y -32.73, Z 98.0, A 0, B 90, C 0} C_DIS
LIN {X -48.26, Y -35.63, Z 98.0, A 0, B 90, C 0} C_DIS
LIN {X -48.08, Y -35.89, Z 98.0, A 0, B 90, C 0} C_DIS
LIN {X -45.88, Y -38.65, Z 98.0, A 0, B 90, C 0} C_DIS
LIN {X -45.69, Y -38.89, Z 98.0, A 0, B 90, C 0} C_DIS
LIN {X -43.31, Y -41.51, Z 98.0, A 0, B 90, C 0} C_DIS
LIN {X -43.1, Y -41.74, Z 98.0, A 0, B 90, C 0} C_DIS
LIN {X -40.56, Y -44.2, Z 98.0, A 0, B 90, C 0} C_DIS
LIN {X -40.34, Y -44.42, Z 98.0, A 0, B 90, C 0} C_DIS
LIN {X -37.64, Y -46.71, Z 98.0, A 0, B 90, C 0} C_DIS
LIN {X -37.41, Y -46.91, Z 98.0, A 0, B 90, C 0} C_DIS
LIN {X -34.57, Y -49.03, Z 98.0, A 0, B 90, C 0} C_DIS
$OUT[1] = FALSE

; END LAYER 48
LIN {X -34.33, Y -49.21, Z 98.0, A 0, B 90, C 0} C_DIS
WAIT SEC 3
LIN {X -34.33, Y -49.21, Z 100.0, A 0, B 90, C 0} C_DIS
$OUT[1] = TRUE
WAIT SEC 0.8
LIN {X -34.33, Y -49.21, Z 100.0, A 0, B 90, C 0} C_DIS
LIN {X -34.33, Y -49.21, Z 100.0, A 0, B 90, C 0} C_DIS
LIN {X -31.23, Y -51.22, Z 100.0, A 0, B 90, C 0} C_DIS
LIN {X -31.1, Y -51.31, Z 100.0, A 0, B 90, C 0} C_DIS
LIN {X -27.89, Y -53.12, Z 100.0, A 0, B 90, C 0} C_DIS
LIN {X -27.75, Y -53.2, Z 100.0, A 0, B 90, C 0} C_DIS
LIN {X -24.43, Y -54.8, Z 100.0, A 0, B 90, C 0} C_DIS
LIN {X -24.29, Y -54.86, Z 100.0, A 0, B 90, C 0} C_DIS
LIN {X -20.86, Y -56.25, Z 100.0, A 0, B 90, C 0} C_DIS
LIN {X -20.72, Y -56.31, Z 100.0, A 0, B 90, C 0} C_DIS
LIN {X -17.22, Y -57.47, Z 100.0, A 0, B 90, C 0} C_DIS
LIN {X -17.07, Y -57.52, Z 100.0, A 0, B 90, C 0} C_DIS
LIN {X -13.5, Y -58.46, Z 100.0, A 0, B 90, C 0} C_DIS
LIN {X -13.35, Y -58.5, Z 100.0, A 0, B 90, C 0} C_DIS
LIN {X -9.73, Y -59.2, Z 100.0, A 0, B 90, C 0} C_DIS
LIN {X -9.58, Y -59.23, Z 100.0, A 0, B 90, C 0} C_DIS
LIN {X -5.91, Y -59.7, Z 100.0, A 0, B 90, C 0} C_DIS
LIN {X -5.76, Y -59.72, Z 100.0, A 0, B 90, C 0} C_DIS
LIN {X -2.08, Y -59.96, Z 100.0, A 0, B 90, C 0} C_DIS
LIN {X -1.92, Y -59.97, Z 100.0, A 0, B 90, C 0} C_DIS
LIN {X 1.77, Y -59.97, Z 100.0, A 0, B 90, C 0} C_DIS
LIN {X 1.92, Y -59.97, Z 100.0, A 0, B 90, C 0} C_DIS
LIN {X 5.61, Y -59.73, Z 100.0, A 0, B 90, C 0} C_DIS
LIN {X 5.76, Y -59.72, Z 100.0, A 0, B 90, C 0} C_DIS
LIN {X 9.42, Y -59.25, Z 100.0, A 0, B 90, C 0} C_DIS
LIN {X 9.58, Y -59.23, Z 100.0, A 0, B 90, C 0} C_DIS
LIN {X 13.2, Y -58.53, Z 100.0, A 0, B 90, C 0} C_DIS
LIN {X 13.35, Y -58.5, Z 100.0, A 0, B 90, C 0} C_DIS
LIN {X 16.92, Y -57.56, Z 100.0, A 0, B 90, C 0} C_DIS
LIN {X 17.07, Y -57.52, Z 100.0, A 0, B 90, C 0} C_DIS
LIN {X 20.58, Y -56.36, Z 100.0, A 0, B 90, C 0} C_DIS
LIN {X 20.72, Y -56.31, Z 100.0, A 0, B 90, C 0} C_DIS
LIN {X 24.14, Y -54.92, Z 100.0, A 0, B 90, C 0} C_DIS
LIN {X 24.29, Y -54.86, Z 100.0, A 0, B 90, C 0} C_DIS
LIN {X 27.61, Y -53.26, Z 100.0, A 0, B 90, C 0} C_DIS
LIN {X 27.75, Y -53.2, Z 100.0, A 0, B 90, C 0} C_DIS
LIN {X 30.97, Y -51.38, Z 100.0, A 0, B 90, C 0} C_DIS
LIN {X 31.1, Y -51.31, Z 100.0, A 0, B 90, C 0} C_DIS
LIN {X 34.2, Y -49.29, Z 100.0, A 0, B 90, C 0} C_DIS
LIN {X 34.33, Y -49.21, Z 100.0, A 0, B 90, C 0} C_DIS
LIN {X 37.29, Y -47.0, Z 100.0, A 0, B 90, C 0} C_DIS
LIN {X 37.41, Y -46.91, Z 100.0, A 0, B 90, C 0} C_DIS
LIN {X 40.22, Y -44.52, Z 100.0, A 0, B 90, C 0} C_DIS
LIN {X 40.34, Y -44.42, Z 100.0, A 0, B 90, C 0} C_DIS
LIN {X 42.99, Y -41.85, Z 100.0, A 0, B 90, C 0} C_DIS
LIN {X 43.1, Y -41.74, Z 100.0, A 0, B 90, C 0} C_DIS
LIN {X 45.58, Y -39.01, Z 100.0, A 0, B 90, C 0} C_DIS
LIN {X 45.69, Y -38.89, Z 100.0, A 0, B 90, C 0} C_DIS
LIN {X 47.99, Y -36.01, Z 100.0, A 0, B 90, C 0} C_DIS
LIN {X 48.08, Y -35.89, Z 100.0, A 0, B 90, C 0} C_DIS
LIN {X 50.2, Y -32.86, Z 100.0, A 0, B 90, C 0} C_DIS
LIN {X 50.29, Y -32.73, Z 100.0, A 0, B 90, C 0} C_DIS
LIN {X 52.2, Y -29.57, Z 100.0, A 0, B 90, C 0} C_DIS
LIN {X 52.28, Y -29.44, Z 100.0, A 0, B 90, C 0} C_DIS
LIN {X 53.99, Y -26.17, Z 100.0, A 0, B 90, C 0} C_DIS
LIN {X 54.06, Y -26.03, Z 100.0, A 0, B 90, C 0} C_DIS
LIN {X 55.55, Y -22.66, Z 100.0, A 0, B 90, C 0} C_DIS
LIN {X 55.62, Y -22.52, Z 100.0, A 0, B 90, C 0} C_DIS
LIN {X 56.89, Y -19.05, Z 100.0, A 0, B 90, C 0} C_DIS
LIN {X 56.94, Y -18.91, Z 100.0, A 0, B 90, C 0} C_DIS
LIN {X 57.99, Y -15.37, Z 100.0, A 0, B 90, C 0} C_DIS
LIN {X 58.04, Y -15.22, Z 100.0, A 0, B 90, C 0} C_DIS
LIN {X 58.86, Y -11.62, Z 100.0, A 0, B 90, C 0} C_DIS
LIN {X 58.89, Y -11.47, Z 100.0, A 0, B 90, C 0} C_DIS
LIN {X 59.48, Y -7.82, Z 100.0, A 0, B 90, C 0} C_DIS
LIN {X 59.51, Y -7.67, Z 100.0, A 0, B 90, C 0} C_DIS
LIN {X 59.86, Y -4.0, Z 100.0, A 0, B 90, C 0} C_DIS
LIN {X 59.88, Y -3.84, Z 100.0, A 0, B 90, C 0} C_DIS
LIN {X 60.0, Y -0.15, Z 100.0, A 0, B 90, C 0} C_DIS
LIN {X 60.0, Y 0.0, Z 100.0, A 0, B 90, C 0} C_DIS
LIN {X 59.88, Y 3.69, Z 100.0, A 0, B 90, C 0} C_DIS
LIN {X 59.88, Y 3.84, Z 100.0, A 0, B 90, C 0} C_DIS
LIN {X 59.52, Y 7.52, Z 100.0, A 0, B 90, C 0} C_DIS
LIN {X 59.51, Y 7.67, Z 100.0, A 0, B 90, C 0} C_DIS
LIN {X 58.92, Y 11.32, Z 100.0, A 0, B 90, C 0} C_DIS
LIN {X 58.89, Y 11.47, Z 100.0, A 0, B 90, C 0} C_DIS
LIN {X 58.07, Y 15.07, Z 100.0, A 0, B 90, C 0} C_DIS
LIN {X 58.04, Y 15.22, Z 100.0, A 0, B 90, C 0} C_DIS
LIN {X 56.99, Y 18.76, Z 100.0, A 0, B 90, C 0} C_DIS
LIN {X 56.94, Y 18.91, Z 100.0, A 0, B 90, C 0} C_DIS
LIN {X 55.67, Y 22.37, Z 100.0, A 0, B 90, C 0} C_DIS
LIN {X 55.62, Y 22.52, Z 100.0, A 0, B 90, C 0} C_DIS
LIN {X 54.12, Y 25.89, Z 100.0, A 0, B 90, C 0} C_DIS
LIN {X 54.06, Y 26.03, Z 100.0, A 0, B 90, C 0} C_DIS
LIN {X 52.35, Y 29.31, Z 100.0, A 0, B 90, C 0} C_DIS
LIN {X 52.28, Y 29.44, Z 100.0, A 0, B 90, C 0} C_DIS
LIN {X 50.37, Y 32.6, Z 100.0, A 0, B 90, C 0} C_DIS
LIN {X 50.29, Y 32.73, Z 100.0, A 0, B 90, C 0} C_DIS
LIN {X 48.17, Y 35.76, Z 100.0, A 0, B 90, C 0} C_DIS
LIN {X 48.08, Y 35.89, Z 100.0, A 0, B 90, C 0} C_DIS
LIN {X 45.78, Y 38.77, Z 100.0, A 0, B 90, C 0} C_DIS
LIN {X 45.69, Y 38.89, Z 100.0, A 0, B 90, C 0} C_DIS
LIN {X 43.2, Y 41.63, Z 100.0, A 0, B 90, C 0} C_DIS
LIN {X 43.1, Y 41.74, Z 100.0, A 0, B 90, C 0} C_DIS
LIN {X 40.45, Y 44.31, Z 100.0, A 0, B 90, C 0} C_DIS
LIN {X 40.34, Y 44.42, Z 100.0, A 0, B 90, C 0} C_DIS
LIN {X 37.53, Y 46.81, Z 100.0, A 0, B 90, C 0} C_DIS
LIN {X 37.41, Y 46.91, Z 100.0, A 0, B 90, C 0} C_DIS
LIN {X 34.45, Y 49.12, Z 100.0, A 0, B 90, C 0} C_DIS
LIN {X 34.33, Y 49.21, Z 100.0, A 0, B 90, C 0} C_DIS
LIN {X 31.23, Y 51.22, Z 100.0, A 0, B 90, C 0} C_DIS
LIN {X 31.1, Y 51.31, Z 100.0, A 0, B 90, C 0} C_DIS
LIN {X 27.89, Y 53.12, Z 100.0, A 0, B 90, C 0} C_DIS
LIN {X 27.75, Y 53.2, Z 100.0, A 0, B 90, C 0} C_DIS
LIN {X 24.43, Y 54.8, Z 100.0, A 0, B 90, C 0} C_DIS
LIN {X 24.29, Y 54.86, Z 100.0, A 0, B 90, C 0} C_DIS
LIN {X 20.86, Y 56.25, Z 100.0, A 0, B 90, C 0} C_DIS
LIN {X 20.72, Y 56.31, Z 100.0, A 0, B 90, C 0} C_DIS
LIN {X 17.22, Y 57.47, Z 100.0, A 0, B 90, C 0} C_DIS
LIN {X 17.07, Y 57.52, Z 100.0, A 0, B 90, C 0} C_DIS
LIN {X 13.5, Y 58.46, Z 100.0, A 0, B 90, C 0} C_DIS
LIN {X 13.35, Y 58.5, Z 100.0, A 0, B 90, C 0} C_DIS
LIN {X 9.73, Y 59.2, Z 100.0, A 0, B 90, C 0} C_DIS
LIN {X 9.58, Y 59.23, Z 100.0, A 0, B 90, C 0} C_DIS
LIN {X 5.91, Y 59.7, Z 100.0, A 0, B 90, C 0} C_DIS
LIN {X 5.76, Y 59.72, Z 100.0, A 0, B 90, C 0} C_DIS
LIN {X 2.08, Y 59.96, Z 100.0, A 0, B 90, C 0} C_DIS
LIN {X 1.92, Y 59.97, Z 100.0, A 0, B 90, C 0} C_DIS
LIN {X -1.77, Y 59.97, Z 100.0, A 0, B 90, C 0} C_DIS
LIN {X -1.92, Y 59.97, Z 100.0, A 0, B 90, C 0} C_DIS
LIN {X -5.61, Y 59.73, Z 100.0, A 0, B 90, C 0} C_DIS
LIN {X -5.76, Y 59.72, Z 100.0, A 0, B 90, C 0} C_DIS
LIN {X -9.42, Y 59.25, Z 100.0, A 0, B 90, C 0} C_DIS
LIN {X -9.58, Y 59.23, Z 100.0, A 0, B 90, C 0} C_DIS
LIN {X -13.2, Y 58.53, Z 100.0, A 0, B 90, C 0} C_DIS
LIN {X -13.35, Y 58.5, Z 100.0, A 0, B 90, C 0} C_DIS
LIN {X -16.92, Y 57.56, Z 100.0, A 0, B 90, C 0} C_DIS
LIN {X -17.07, Y 57.52, Z 100.0, A 0, B 90, C 0} C_DIS
LIN {X -20.58, Y 56.36, Z 100.0, A 0, B 90, C 0} C_DIS
LIN {X -20.72, Y 56.31, Z 100.0, A 0, B 90, C 0} C_DIS
LIN {X -24.14, Y 54.92, Z 100.0, A 0, B 90, C 0} C_DIS
LIN {X -24.29, Y 54.86, Z 100.0, A 0, B 90, C 0} C_DIS
LIN {X -27.61, Y 53.26, Z 100.0, A 0, B 90, C 0} C_DIS
LIN {X -27.75, Y 53.2, Z 100.0, A 0, B 90, C 0} C_DIS
LIN {X -30.97, Y 51.38, Z 100.0, A 0, B 90, C 0} C_DIS
LIN {X -31.1, Y 51.31, Z 100.0, A 0, B 90, C 0} C_DIS
LIN {X -34.2, Y 49.29, Z 100.0, A 0, B 90, C 0} C_DIS
LIN {X -34.33, Y 49.21, Z 100.0, A 0, B 90, C 0} C_DIS
LIN {X -37.29, Y 47.0, Z 100.0, A 0, B 90, C 0} C_DIS
LIN {X -37.41, Y 46.91, Z 100.0, A 0, B 90, C 0} C_DIS
LIN {X -40.22, Y 44.52, Z 100.0, A 0, B 90, C 0} C_DIS
LIN {X -40.34, Y 44.42, Z 100.0, A 0, B 90, C 0} C_DIS
LIN {X -42.99, Y 41.85, Z 100.0, A 0, B 90, C 0} C_DIS
LIN {X -43.1, Y 41.74, Z 100.0, A 0, B 90, C 0} C_DIS
LIN {X -45.58, Y 39.01, Z 100.0, A 0, B 90, C 0} C_DIS
LIN {X -45.69, Y 38.89, Z 100.0, A 0, B 90, C 0} C_DIS
LIN {X -47.99, Y 36.01, Z 100.0, A 0, B 90, C 0} C_DIS
LIN {X -48.08, Y 35.89, Z 100.0, A 0, B 90, C 0} C_DIS
LIN {X -50.2, Y 32.86, Z 100.0, A 0, B 90, C 0} C_DIS
LIN {X -50.29, Y 32.73, Z 100.0, A 0, B 90, C 0} C_DIS
LIN {X -52.2, Y 29.57, Z 100.0, A 0, B 90, C 0} C_DIS
LIN {X -52.28, Y 29.44, Z 100.0, A 0, B 90, C 0} C_DIS
LIN {X -53.99, Y 26.17, Z 100.0, A 0, B 90, C 0} C_DIS
LIN {X -54.06, Y 26.03, Z 100.0, A 0, B 90, C 0} C_DIS
LIN {X -55.55, Y 22.66, Z 100.0, A 0, B 90, C 0} C_DIS
LIN {X -55.62, Y 22.52, Z 100.0, A 0, B 90, C 0} C_DIS
LIN {X -56.89, Y 19.05, Z 100.0, A 0, B 90, C 0} C_DIS
LIN {X -56.94, Y 18.91, Z 100.0, A 0, B 90, C 0} C_DIS
LIN {X -57.99, Y 15.37, Z 100.0, A 0, B 90, C 0} C_DIS
LIN {X -58.04, Y 15.22, Z 100.0, A 0, B 90, C 0} C_DIS
LIN {X -58.86, Y 11.62, Z 100.0, A 0, B 90, C 0} C_DIS
LIN {X -58.89, Y 11.47, Z 100.0, A 0, B 90, C 0} C_DIS
LIN {X -59.48, Y 7.82, Z 100.0, A 0, B 90, C 0} C_DIS
LIN {X -59.51, Y 7.67, Z 100.0, A 0, B 90, C 0} C_DIS
LIN {X -59.86, Y 4.0, Z 100.0, A 0, B 90, C 0} C_DIS
LIN {X -59.88, Y 3.84, Z 100.0, A 0, B 90, C 0} C_DIS
LIN {X -60.0, Y 0.15, Z 100.0, A 0, B 90, C 0} C_DIS
LIN {X -60.0, Y -0.0, Z 100.0, A 0, B 90, C 0} C_DIS
LIN {X -59.88, Y -3.69, Z 100.0, A 0, B 90, C 0} C_DIS
LIN {X -59.88, Y -3.84, Z 100.0, A 0, B 90, C 0} C_DIS
LIN {X -59.52, Y -7.52, Z 100.0, A 0, B 90, C 0} C_DIS
LIN {X -59.51, Y -7.67, Z 100.0, A 0, B 90, C 0} C_DIS
LIN {X -58.92, Y -11.32, Z 100.0, A 0, B 90, C 0} C_DIS
LIN {X -58.89, Y -11.47, Z 100.0, A 0, B 90, C 0} C_DIS
LIN {X -58.07, Y -15.07, Z 100.0, A 0, B 90, C 0} C_DIS
LIN {X -58.04, Y -15.22, Z 100.0, A 0, B 90, C 0} C_DIS
LIN {X -56.99, Y -18.76, Z 100.0, A 0, B 90, C 0} C_DIS
LIN {X -56.94, Y -18.91, Z 100.0, A 0, B 90, C 0} C_DIS
LIN {X -55.67, Y -22.37, Z 100.0, A 0, B 90, C 0} C_DIS
LIN {X -55.62, Y -22.52, Z 100.0, A 0, B 90, C 0} C_DIS
LIN {X -54.12, Y -25.89, Z 100.0, A 0, B 90, C 0} C_DIS
LIN {X -54.06, Y -26.03, Z 100.0, A 0, B 90, C 0} C_DIS
LIN {X -52.35, Y -29.31, Z 100.0, A 0, B 90, C 0} C_DIS
LIN {X -52.28, Y -29.44, Z 100.0, A 0, B 90, C 0} C_DIS
LIN {X -50.37, Y -32.6, Z 100.0, A 0, B 90, C 0} C_DIS
LIN {X -50.29, Y -32.73, Z 100.0, A 0, B 90, C 0} C_DIS
LIN {X -48.17, Y -35.76, Z 100.0, A 0, B 90, C 0} C_DIS
LIN {X -48.08, Y -35.89, Z 100.0, A 0, B 90, C 0} C_DIS
LIN {X -45.78, Y -38.77, Z 100.0, A 0, B 90, C 0} C_DIS
LIN {X -45.69, Y -38.89, Z 100.0, A 0, B 90, C 0} C_DIS
LIN {X -43.2, Y -41.63, Z 100.0, A 0, B 90, C 0} C_DIS
LIN {X -43.1, Y -41.74, Z 100.0, A 0, B 90, C 0} C_DIS
LIN {X -40.45, Y -44.31, Z 100.0, A 0, B 90, C 0} C_DIS
LIN {X -40.34, Y -44.42, Z 100.0, A 0, B 90, C 0} C_DIS
LIN {X -37.53, Y -46.81, Z 100.0, A 0, B 90, C 0} C_DIS
LIN {X -37.41, Y -46.91, Z 100.0, A 0, B 90, C 0} C_DIS
LIN {X -34.45, Y -49.12, Z 100.0, A 0, B 90, C 0} C_DIS
$OUT[1] = FALSE

; END LAYER 49
;END USER CODE
;HOME
;FOLD PTP HOME Vel=10% DEFAULT
$BWDSTART=FALSE
$H_POS=XHOME
PDAT_ACT=PDEFAULT
FDAT_ACT=FHOME
BAS(#PTP_DAT )
BAS (#VEL_PTP,10 )
PTP XHOME
;ENDFOLD
END

--- cilindro.dat ---
DEFDAT cilindro()
ENDDAT
